FUNCTION_BLOCK FB_EXT_TREATY_VGC
VAR_INPUT
    TREATY_VGC : ST_VGC;
END_VAR
VAR_OUTPUT
END_VAR
VAR
    q_xTREATY_VGC_STATUS AT%Q*: BOOL;
END_VAR

q_xTREATY_VGC_STATUS := TREATY_VGC.eState = E_ValvePositionState.OPEN;

END_FUNCTION_BLOCK

(* stored: Version 1.1.0.1, ProductVersion 3.1.4024.2
   POU FB_EXT_TREATY_VGC: Id {cc8265de-575f-4e4a-be6e-e4d049fa76c4}, SpecialFunc None *)
